// TIA Portal V17 program export: 1 tag tables, 0 data types, 0 data blocks, 3 code blocks (in call order from the OBs), 3 instance data blocks

VAR_GLOBAL   // PLC tag table "Default tag table"
   AX_4_Actor_Interface_AddressIn AT %I356.0 : "PD_TEL105_IN";
   AX_4_Actor_Interface_AddressOut AT %Q356.0 : "PD_TEL105_OUT";
   AX_4_Actor_Interface_TorqueDataAddressIn AT %I382.0 : "PD_TEL750_IN";
   AX_4_Actor_Interface_TorqueDataAddressOut AT %Q382.0 : "PD_TEL750_OUT";
   AX_3_Actor_Interface_AddressIn AT %I324.0 : "PD_TEL105_IN";
   AX_3_Actor_Interface_AddressOut AT %Q324.0 : "PD_TEL105_OUT";
   AX_3_Actor_Interface_TorqueDataAddressIn AT %I350.0 : "PD_TEL750_IN";
   AX_3_Actor_Interface_TorqueDataAddressOut AT %Q350.0 : "PD_TEL750_OUT";
   AX_2_Actor_Interface_AddressIn AT %I292.0 : "PD_TEL105_IN";
   AX_2_Actor_Interface_AddressOut AT %Q292.0 : "PD_TEL105_OUT";
   AX_2_Actor_Interface_TorqueDataAddressIn AT %I318.0 : "PD_TEL750_IN";
   AX_2_Actor_Interface_TorqueDataAddressOut AT %Q318.0 : "PD_TEL750_OUT";
   AX_1_Actor_Interface_AddressIn AT %I260.0 : "PD_TEL105_IN";
   AX_1_Actor_Interface_AddressOut AT %Q260.0 : "PD_TEL105_OUT";
   AX_1_Actor_Interface_TorqueDataAddressIn AT %I286.0 : "PD_TEL750_IN";
   AX_1_Actor_Interface_TorqueDataAddressOut AT %Q286.0 : "PD_TEL750_OUT";
   SpeedAxis_Actor_Interface_AddressIn AT %I288.0 : "PD_TEL1_IN";
   SpeedAxis_Actor_Interface_AddressOut AT %Q390.0 : "PD_TEL1_OUT";
   Tag_1 AT %M0.0 : Bool;
   Tag_2 AT %M0.1 : Bool;
   Tag_3 AT %M0.2 : Bool;
   Tag_4 AT %M0.3 : Bool;
END_VAR

ORGANIZATION_BLOCK "Main"   // OB1, LAD, ProgramCycle
TITLE = "Main Program Sweep (Cycle)"
{ S7_Optimized_Access := 'TRUE' }
VERSION : 0.1
// stored: AutoNumber true, IsIECCheckEnabled false, SetENOAutomatically false
   VAR_INPUT
      Initial_Call : Bool;   // Initial call of this OB
      Remanence : Bool;   // =True, if remanent data are available
   END_VAR
BEGIN

REGION Network 1
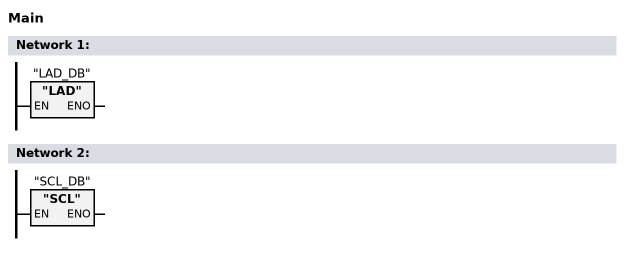
   RUNG wire#powerrail
      "LAD_DB"()
   END_RUNG
   // the same network as SCL:
   "LAD_DB"();   // "LAD"
END_REGION

REGION Network 2
   RUNG wire#powerrail
      "SCL_DB"()
   END_RUNG
   // the same network as SCL:
   "SCL_DB"();   // "SCL"
END_REGION
END_ORGANIZATION_BLOCK

FUNCTION_BLOCK "Test_VCI"   // FB2, LAD
{ S7_Optimized_Access := 'TRUE' }
VERSION : 0.1
// stored: AutoNumber true, IsIECCheckEnabled false, IsRetainMemResEnabled false, MemoryReserve 100, SetENOAutomatically false, UDAEnableTagReadback false
   VAR_INPUT
      In : Bool;
   END_VAR
   VAR_OUTPUT
      Out : Bool;
   END_VAR
BEGIN

REGION Network 1
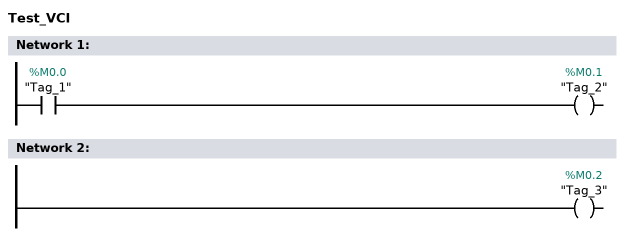
   RUNG wire#powerrail
      Contact( "Tag_1" )
      Coil( "Tag_2" )
   END_RUNG
   // the same network as SCL:
   "Tag_2" := "Tag_1";
END_REGION

REGION Network 2
   RUNG wire#powerrail
      Coil( "Tag_3" )
   END_RUNG
   // the same network as SCL:
   "Tag_3" := TRUE;
END_REGION
END_FUNCTION_BLOCK

FUNCTION_BLOCK "Main_Safety_RTG1"   // FB1, F_FBD
{ S7_Optimized_Access := 'TRUE' }
VERSION : 0.1
// stored: AutoNumber false, IsIECCheckEnabled false, UDAEnableTagReadback false
BEGIN
END_FUNCTION_BLOCK

DATA_BLOCK "Test_VCI_DB"   // DB8
VERSION : 0.1
// stored: AutoNumber true, DBAccessibleFromOPCUA true, DBAccessibleFromWebserver true, InstanceOfName Test_VCI, InstanceOfType FB
"Test_VCI"
BEGIN
END_DATA_BLOCK

DATA_BLOCK "Test_VCI_DB_1"   // DB9
VERSION : 0.1
// stored: AutoNumber true, DBAccessibleFromOPCUA true, DBAccessibleFromWebserver true, InstanceOfName Test_VCI, InstanceOfType FB
"Test_VCI"
BEGIN
END_DATA_BLOCK

DATA_BLOCK "Main_Safety_RTG1_DB"   // DB6, F_DB
NAME : FUSI
VERSION : 0.1
// stored: AutoNumber true, DBAccessibleFromOPCUA true, DBAccessibleFromWebserver true, InstanceOfName Main_Safety_RTG1, InstanceOfType FB
"Main_Safety_RTG1"
BEGIN
END_DATA_BLOCK
